Staubli VAL3: Form_Panel.pgx

public program Form_Panel(string x_sTitle, string x_sPanelTitle, num& x_nSelectIndex, string x_sBottom)
begin

cls()
title(x_sTitle)
call Control_LeftS(x_sBottom)
call Control_PanelXY(22,0,15,10)
call Control_Panel(x_sPanelTitle)
call Control_BottomS(x_sBottom)


//call Control_List(x_sList,x_nSelectIndex)



end
